TYPE ST_PMPS_Attenuator : 
    STRUCT
        nReqAtt : UINT;
        nAttCur : UINT;
        xAttOK : UINT;
    END_STRUCT
END_TYPE

(* stored: Version 1.1.0.1, ProductVersion 3.1.4024.0
   DUT ST_PMPS_Attenuator: Id {cd9a5cb4-772a-4c5d-92cc-8611a9fb1859} *)
